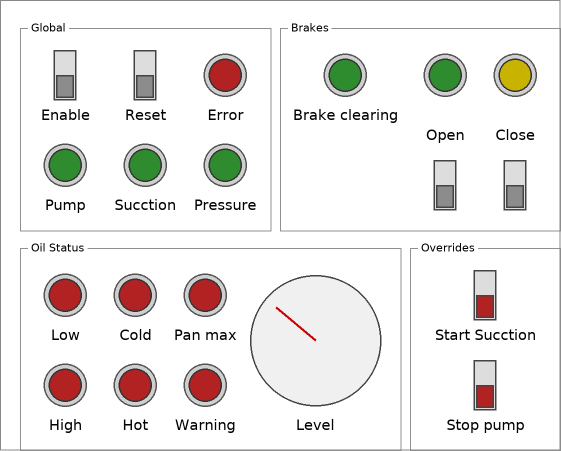
VISUALIZATION Hydraulics  // 561x451
    GroupBox (20,20 251x211), "Global"
        DipSwitch (20,30 50x50), variable: MAIN.HydraulicsControl.enable, behaviour: TOGGLE, style: Switch-DipSwitch-Gray
        DipSwitch (100,30 50x50), variable: MAIN.HydraulicsControl.reset, behaviour: TOGGLE, style: Switch-DipSwitch-Gray
        Label (0,80 91x30), "Enable"
        Label (90,80 71x30), "Reset"
        Lamp1 (180,30 50x50), variable: MAIN.HydraulicsControl.error, style: Lamp-Lamp1-Red
        Label (180,80 51x30), "Error"
        Lamp1 (20,120 50x50), variable: MAIN.HydraulicsControl.pump_running, style: Lamp-Lamp1-Green
        Lamp1 (100,120 50x50), variable: MAIN.HydraulicsControl.suction_running, style: Lamp-Lamp1-Green
        Lamp1 (180,120 50x50), variable: MAIN.HydraulicsControl.oil_pressure_OK, style: Lamp-Lamp1-Green
        Label (20,170 51x30), "Pump"
        Label (90,170 71x30), "Sucction"
        Label (170,170 71x30), "Pressure"
    GroupBox (280,20 281x211), "Brakes"
        DipSwitch (140,140 50x50), variable: MAIN.HydraulicsControl.iopen_brake, behaviour: TOGGLE, style: Switch-DipSwitch-Gray
        Label (130,100 71x30), "Open"
        Label (10,80 111x30), "Brake clearing"
        Lamp1 (40,30 50x50), variable: MAIN.HydraulicsControl.brake_clearing, style: Lamp-Lamp1-Green
        DipSwitch (210,140 50x50), variable: MAIN.HydraulicsControl.iclose_brake, behaviour: TOGGLE, style: Switch-DipSwitch-Gray
        Label (210,100 51x30), "Close"
        Lamp1 (140,30 50x50), variable: MAIN.HydraulicsControl.brake_open, style: Lamp-Lamp1-Green
        Lamp1 (210,30 50x50), variable: MAIN.HydraulicsControl.brake_closed, style: Lamp-Lamp1-Yellow
    GroupBox (410,240 151x211), "Overrides"
        DipSwitch (50,30 50x50), variable: MAIN.HydraulicsControl.suction_manual, behaviour: TOGGLE, style: Switch-DipSwitch-Red
        DipSwitch (50,120 50x50), variable: MAIN.HydraulicsControl.pump_manual_stop, behaviour: TOGGLE, style: Switch-DipSwitch-Red
        Label (20,80 111x30), "Start Sucction"
        Label (30,170 91x30), "Stop pump"
    GroupBox (20,240 381x211), "Oil Status"
        Lamp1 (20,30 50x50), variable: MAIN.HydraulicsControl.oil_low, style: Lamp-Lamp1-Red
        Label (20,80 51x30), "Low"
        Lamp1 (20,120 50x50), variable: MAIN.HydraulicsControl.oil_high, style: Lamp-Lamp1-Red
        Label (10,170 71x30), "High"
        Lamp1 (160,120 50x50), variable: MAIN.HydraulicsControl.oil_warning, style: Lamp-Lamp1-Red
        Label (150,170 71x30), "Warning"
        Lamp1 (90,30 50x50), variable: MAIN.HydraulicsControl.oil_cold, style: Lamp-Lamp1-Red
        Label (90,80 51x30), "Cold"
        Lamp1 (90,120 50x50), variable: MAIN.HydraulicsControl.oil_hot, style: Lamp-Lamp1-Red
        Label (90,170 51x30), "Hot"
        Lamp1 (160,30 50x50), variable: MAIN.HydraulicsControl.oilpan_maximum, style: Lamp-Lamp1-Red
        Label (140,80 91x30), "Pan max"
        Meter360 (230,30 131x141), value: MAIN.HydraulicsControl.oil_level, style: Meter-Meter360-Gray, scale format: %.0f%, scale 0..120
        Label (260,170 71x30), "Level"
END_VISUALIZATION

(* stored: Version 1.1.0.1, ProductVersion 3.1.4026.8
   Visu Hydraulics: Id {371113af-a8cf-42ba-8f72-dc02b3afe399} *)
